FUNCTION ScaleTrans_1 : REAL
VAR_INPUT
	EN:BOOL;//启动条件
	Scalln:REAL;//输入值
	X0:REAL;//输入范围下限值
	Y0:REAL;//输出范围下限值
	X1:REAL;//输入范围上限值
	Y1:REAL;//输出范围上限值
	Sclofs:REAL;//偏置值
END_VAR
VAR
END_VAR

IF EN THEN
	IF (X1-X0)<> 0 THEN
		ScaleTrans:=(Y1-Y0)/(X1-X0)*(Scalln-X0)+Y0+Sclofs;
	END_IF
END_IF

END_FUNCTION

(* stored: Version 1.1.0.1, ProductVersion 3.1.4024.9
   POU ScaleTrans_1: Id {ec8dfced-4476-429e-b8ac-f2b38599c5d8}, SpecialFunc None *)
